// TIA Portal project "CANPACK_CPD" (V19)

(* hardware
DEVICE "S7-1500/ET200MP station_1"  S7-1500 station
   slot 0: "Rail_0"  Rack  6ES7 590-1***0-0AA0
   slot 1: "PLC_1"  CPU 1511F-1 PN  6ES7 511-1FL03-0AB0  V3.1
      slot 3: "CPU display_1"  6ES7591-1AA00-0AA0
      slot 32768: "PROFINET interface_1"  X1
         slot 32769: "Port_1"  X1 P1
         slot 32770: "Port_2"  X1 P2
      slot 34817: "Virtual CP interface port_1"  Virtual CP interface port  Virtual CP interface port
*)

// ===== PLC "PLC_1"  CPU 1511F-1 PN =====
// protected blocks, not shown: "Main_Safety_RTG1", "Main_Safety_RTG1_DB"

VAR_GLOBAL   // PLC tag table "Default tag table"
   "Clock_Byte" AT %MB0 : Byte;
   "Clock_10Hz" AT %M0.0 : Bool;
   "Clock_5Hz" AT %M0.1 : Bool;
   "Clock_2.5Hz" AT %M0.2 : Bool;
   "Clock_2Hz" AT %M0.3 : Bool;
   "Clock_1.25Hz" AT %M0.4 : Bool;
   "Clock_1Hz" AT %M0.5 : Bool;
   "Clock_0.625Hz" AT %M0.6 : Bool;
   "Clock_0.5Hz" AT %M0.7 : Bool;
END_VAR

DATA_BLOCK "DATA"   // DB3
{ S7_Optimized_Access := 'TRUE' }
VERSION : 0.1
   VAR
      connection : TCON_IP_v4;
      value : UInt;
      activate : Bool;
      status1 : UInt;
      velocity1 : UInt;
      status2 : UInt;
      velocity2 : UInt;
      state : Int;
   END_VAR
BEGIN
   connection.InterfaceId := 64;
   connection.ID := 1;
   connection.ActiveEstablished := 1;
   connection.RemoteAddress.ADDR[1] := 192;
   connection.RemoteAddress.ADDR[2] := 168;
   connection.RemoteAddress.ADDR[3] := 0;
   connection.RemoteAddress.ADDR[4] := 10;
   connection.RemotePort := 20001;
   connection.LocalPort := 20001;
END_DATA_BLOCK

// folder: System blocks/Program resources

DATA_BLOCK "IEC_Counter_0_DB"   // DB4
{ S7_Optimized_Access := 'TRUE' }
AUTHOR : Simatic
FAMILY : IEC
NAME : CNTR
VERSION : 1.0
// stored: InstanceOfName IEC_COUNTER
"IEC_COUNTER"
BEGIN
END_DATA_BLOCK

// folder: (top level)

ORGANIZATION_BLOCK "Main"   // OB1, LAD, ProgramCycle
TITLE = "Main Program Sweep (Cycle)"
{ S7_Optimized_Access := 'TRUE' }
VERSION : 0.1
   VAR_INPUT
      Initial_Call : Bool;   // Initial call of this OB
      Remanence : Bool;   // =True, if remanent data are available
   END_VAR
BEGIN

REGION Network 1
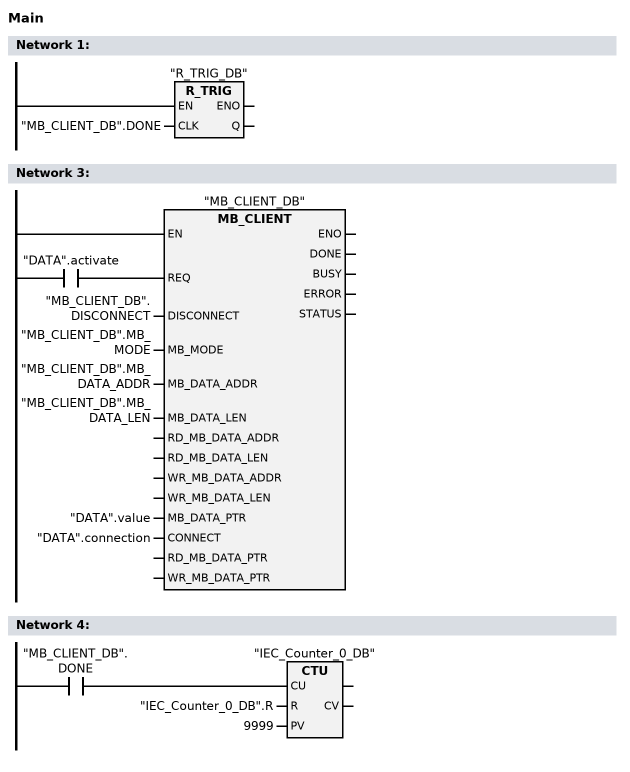
   "R_TRIG_DB"(CLK := "MB_CLIENT_DB".DONE);   // R_TRIG
END_REGION

REGION Network 2 (SCL)
   CASE "DATA".state OF
       0:
           "DATA".activate := 1;
           "MB_CLIENT_DB".MB_MODE := 0;
           "MB_CLIENT_DB".MB_DATA_ADDR := 48451;
           "MB_CLIENT_DB".MB_DATA_LEN := 1;
           "MB_CLIENT_DB".MB_Unit_ID := 1;

           IF "R_TRIG_DB".Q THEN
               "DATA".activate := 0;
               "DATA".status1 := "DATA".value;
               "DATA".state := 10;
           END_IF;

       10:
           "DATA".activate := 1;
           "MB_CLIENT_DB".MB_MODE := 1;
           "MB_CLIENT_DB".MB_DATA_ADDR := 48194;
           "MB_CLIENT_DB".MB_DATA_LEN := 1;
           "MB_CLIENT_DB".MB_Unit_ID := 1;
           "DATA".value := "DATA".velocity1;

           IF "R_TRIG_DB".Q THEN
               "DATA".velocity1 := "DATA".velocity1 + 100;
               "DATA".activate := 0;
               "DATA".state := 20;
           END_IF;

       20:
           "DATA".activate := 1;
           "MB_CLIENT_DB".MB_MODE := 0;
           "MB_CLIENT_DB".MB_DATA_ADDR := 48451;
           "MB_CLIENT_DB".MB_DATA_LEN := 1;
           "MB_CLIENT_DB".MB_Unit_ID := 2;

           IF "R_TRIG_DB".Q THEN
               "DATA".activate := 0;
               "DATA".status2 := "DATA".value;
               "DATA".state := 30;
           END_IF;

       30:
           "DATA".activate := 1;
           "MB_CLIENT_DB".MB_MODE := 1;
           "MB_CLIENT_DB".MB_DATA_ADDR := 48194;
           "MB_CLIENT_DB".MB_DATA_LEN := 1;
           "MB_CLIENT_DB".MB_Unit_ID := 2;
           "DATA".value := "DATA".velocity2;

           IF "R_TRIG_DB".Q THEN
               "DATA".velocity2 := "DATA".velocity2 + 100;
               "DATA".activate := 0;
               "DATA".state := 0;
           END_IF;
   END_CASE;

   IF "DATA".velocity1 > 4000 THEN
       "DATA".velocity1 := 100;
   END_IF;
   IF "DATA".velocity2 > 4000 THEN
       "DATA".velocity2 := 100;
   END_IF;
END_REGION

REGION Network 3
   "MB_CLIENT_DB"(REQ := "DATA".activate,   // MB_CLIENT
                  DISCONNECT := "MB_CLIENT_DB".DISCONNECT,
                  MB_MODE := "MB_CLIENT_DB".MB_MODE,
                  MB_DATA_ADDR := "MB_CLIENT_DB".MB_DATA_ADDR,
                  MB_DATA_LEN := "MB_CLIENT_DB".MB_DATA_LEN,
                  MB_DATA_PTR := "DATA".value,
                  CONNECT := "DATA".connection);
END_REGION

REGION Network 4
   "IEC_Counter_0_DB".CTU(CU := "MB_CLIENT_DB".DONE, R := "IEC_Counter_0_DB".R, PV := 9999);
END_REGION
END_ORGANIZATION_BLOCK